// TIA Portal V16 export
// export: Created 2023-08-28T09:37:43.1797762Z, ExportSetting WithDefaults, DisplayName Totally Integrated Automation Portal, DisplayVersion V16 Update 6, DisplayName TIA Portal Version Control Interface, DisplayVersion V16 Update 2, DisplayName TIA Portal Openness, DisplayVersion V16 Update 6, DisplayName STEP 7 Professional, DisplayVersion V16 Update 6, DisplayName STEP 7 Safety, DisplayVersion V16, DisplayName WinCC Advanced, DisplayVersion V16 Update 6
DATA_BLOCK "FindPumpWithMinWorkTime_DB_1"   // DB87
AUTHOR : rtecmer
VERSION : 0.1
// stored: AutoNumber true, DBAccessibleFromOPCUA true, InstanceOfName FindPumpWithMinWorkTime, InstanceOfType FB
"FindPumpWithMinWorkTime"
   // VAR_IN_OUT
   //    chosenPump : Int;
   // END_VAR
   // VAR
   //    minTime : Real;
   // END_VAR
BEGIN
END_DATA_BLOCK
